PROGRAM MAIN
VAR

END_VAR

(*Ethercat Diagnostics*)
DIAGNOSTICS();



(* Call all Programs*)
PRG_ILK();
PRG_DIFF_PUMP();
PRG_ROOTS();
PRG_GATT();
PRG_GEM();

END_PROGRAM

(* stored: Version 1.1.0.1, ProductVersion 3.1.4022.16
   POU MAIN: Id {45381f7c-4c5f-4ec8-9129-311fb837ab4d}, SpecialFunc None *)
